FUNCTION_BLOCK FB_Manual
VAR_INPUT
END_VAR
VAR_OUTPUT
END_VAR
VAR
END_VAR

END_FUNCTION_BLOCK

(* stored: Version 1.1.0.1, ProductVersion 3.1.4024.13
   POU FB_Manual: Id {47b8b6cb-7452-434b-a087-5026a0bf9b80}, SpecialFunc None *)
